// TwinCAT 3 PLC project Woche04
// ProgramVersion: 3.1.4023.0
// libraries:
//   Tc2_Standard, * (Beckhoff Automation GmbH)
//   Tc2_System, * (Beckhoff Automation GmbH)
//   Tc3_Module, * (Beckhoff Automation GmbH)
//   VisuSymbols,3.5.10.0,System
// project tree:
//   DUTs/ ST_MotorValues.TcDUT
//   / GlobalTextList.TcGTLO, PlcTask.TcTTO, Task_4.TcTTO, Visualisierungsmanager.TcVMO (not stored)
//   POUs/ FB_counter.TcPOU, MAIN.TcPOU, F_counter.TcPOU, F_MotorCalc.TcPOU, P_counter.TcPOU
//   VISUs/ Visualization.TcVIS
// real-time tasks:
//   TASK PlcTask: cycle T#10ms, priority 20, ADS port 350
//   TASK Task 4: cycle T#20ms, priority 1, ADS port 351

CONFIGURATION Woche04
    RESOURCE PLC ON TwinCAT3
        TASK PlcTask(INTERVAL := T#10ms, PRIORITY := 20);
        TASK Task_4(INTERVAL := T#20ms, PRIORITY := 1);
        PROGRAM MAIN WITH PlcTask : MAIN;
        PROGRAM P_counter WITH PlcTask : P_counter;
        PROGRAM P_counter WITH Task_4 : P_counter;
    END_RESOURCE
END_CONFIGURATION

// ---- DUTs/ST_MotorValues.TcDUT
TYPE ST_MotorValues :
STRUCT
	iEncoderPosition 	: INT;
	rSpeed				: REAL;
	bOverheat			: BOOL;
END_STRUCT
END_TYPE

// ---- POUs/MAIN.TcPOU
PROGRAM MAIN
VAR
	iCounter 		: INT := 0;
	fb_counter1 	: FB_counter;
	fb_counter2 	: FB_counter;
	iCounterOutFb2 	: INT; 
	
	f_counter1 		: INT;
	
	(*-------------------------------------------*)

	st_motorValues 	: ST_MotorValues; 
	
	rtest1 			: REAL;
	rtest2 			: REAL;
	rtest3 			: REAL;
	
	(* Timer*) 
	ton_timer1 		: Ton;
	btimer_start	: BOOL;
	bLamp 			: bool;
	
END_VAR


(*------------------- Counter als PRG, Fkt und FB ------------------------*)

iCounter := iCounter +1; // Referenz counter im Main

(* Counter Aufruf in einem Programm*) 
P_counter();
P_counter(); // wird 2 mal aufgerufen im Main und einmal im Task_4 

(* Counter Aufruf als Funktionsbausteine *)
fb_counter1(iCounterStep := 1); // Erste Instanz des Counter FBs: Aufruf mit Schrittweite 1
fb_counter1(iCounterStep := 2); // aufruf mit Schrittweite 2


fb_counter1.iCounterStep := 3; 
fb_counter1(); // ist äquivalient zu: fb_counter1(iCounterStep := 3);

fb_counter2(); // zweite Instanz des Counter FBs

fb_counter2(iCounterOut => iCounterOutFb2);  // Counterwerte output wird einer Variable im Main zugewiesen (inkl. Aufruf)  
iCounterOutFb2 := fb_counter2.iCounterOut;  // Counterwerte output wird einer Variable im Main zugewiesen (ohne. Aufruf)

(* Counter Aufruf als Funktion *)
// Hat kein Gedächtnis, counter Zwischenresultat wird deshalb im Main (in Variable f_counter1) gespeichert
f_counter1 := F_counter(iCounter := f_counter1, iCounterStep := 2); 


(*-------------------Funktion mit struct als Returnwert ------------------------*)
st_motorValues := F_MotorCalc();


(*------------------- Typenkonvertiertung ------------------------*)
rtest1 := 10/3;
rtest2 := 10/3.0;
rtest3 := 10/INT_TO_REAL(3);


(*------------------- Timer ------------------------*)
// Timeraufruf Variante 1
ton_timer1(IN := btimer_start, PT:= T#5S);


// Timeraufruf Variante 2
ton_timer1.IN := btimer_start;
ton_timer1.PT:= T#5S;
ton_timer1();

IF ton_timer1.Q THEN // Code für Blinkelampe
	ton_timer1(IN:=FALSE);
	bLamp := NOT(bLamp);
END_IF

END_PROGRAM

// ---- POUs/FB_counter.TcPOU
FUNCTION_BLOCK FB_counter
VAR_INPUT
	iCounterStep : INT := 1;
END_VAR
VAR_OUTPUT
	iCounterOut : INT;
END_VAR
VAR
	iCounter : INT := 0;
END_VAR

iCounter := iCounter + iCounterStep;

END_FUNCTION_BLOCK

// ---- POUs/P_counter.TcPOU
PROGRAM P_counter
VAR
	iCounter : INT := 0;
END_VAR

iCounter := iCounter +1;

END_PROGRAM

// ---- POUs/F_counter.TcPOU
FUNCTION F_counter : INT
VAR_INPUT
	iCounter : INT := 0;
	iCounterStep : INT;
END_VAR
VAR

END_VAR

iCounter := iCounter +iCounterStep;

F_counter := iCounter;

END_FUNCTION

// ---- POUs/F_MotorCalc.TcPOU
FUNCTION F_MotorCalc : ST_MotorValues
VAR_INPUT
END_VAR
VAR
END_VAR


F_MotorCalc.bOverheat := TRUE;
F_MotorCalc.iEncoderPosition := 485;

END_FUNCTION

// ---- VISUs/Visualization.TcVIS
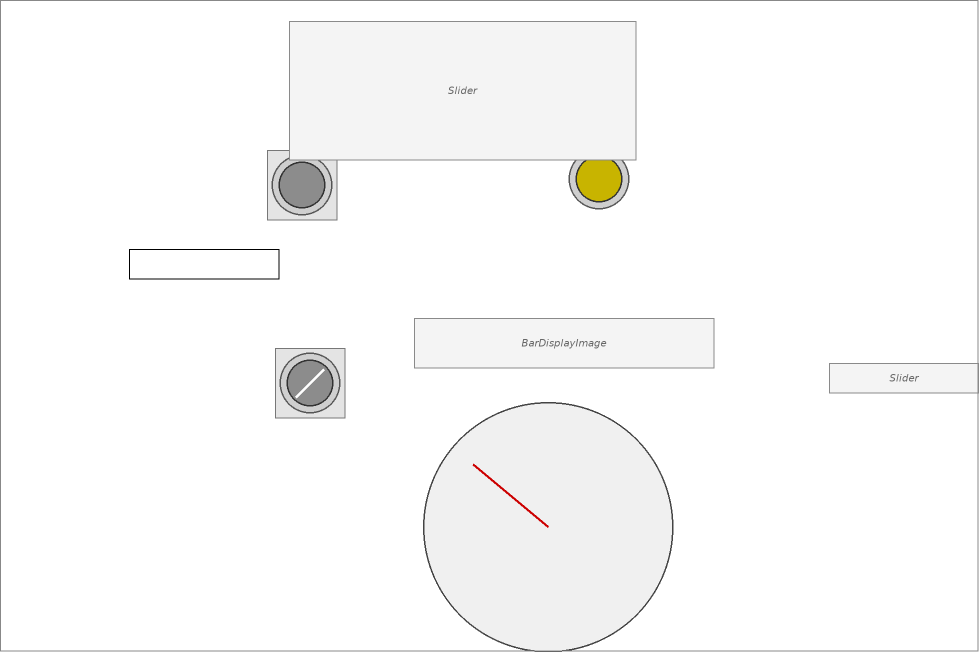
VISUALIZATION Visualization  // 979x652
    Lamp1 (564,144 70x70), variable: MAIN.bLamp, style: Lamp-Lamp1-Yellow
    PushSwitchLed (267,150 70x70), variable: MAIN.btimer_start, behaviour: TOGGLE, style: Switch-PushSwitchLed-Gray
    RotarySwitch (275,348 70x70), behaviour: TOGGLE, style: Switch-RotarySwitch-Gray
    BarDisplayImage (414,318 300x50), value: MAIN.iCounter, style: BarDisplayImage-Gray, scale format: %.1f, scale 0..100
    Meter180 (423,402 250x250), style: Meter-Meter180-Gray, scale format: %.1f, scale 0..100
    Rectangle (129,249 150x30)
    Slider (289,21 347x139), scale 0..1200
    Slider (829,363 150x30), scale 0..100
END_VISUALIZATION
